FUNCTION Convert_TOD_TO_DATE : BOOL
VAR_INPUT
	in : TOD;
	out : REFERENCE TO DATE;
END_VAR
VAR
	converted : DATE;
END_VAR

converted := TOD_TO_DATE(in);

IF (DATE_TO_TOD(converted) <> in) THEN
	RETURN;
END_IF

out := converted;
Convert_TOD_TO_DATE := TRUE;

END_FUNCTION

(* stored: Version 1.1.0.1, ProductVersion 3.1.4024.12
   POU Convert_TOD_TO_DATE: Id {a5c1dcdb-b2b8-4044-8458-c9c919997faf}, SpecialFunc None *)
